DEVICE_TYPE RMT_PRXY (* Proxy for a Remotely Managed Device *)
  (* Standard: 61499 ITA; Description: Remotely Managed Device Proxy *)
  (* Version 0.2, 2002-01-01, JHC, Rockwell Automation, Added WAIT input. *)
  (* Version 0.1, 2001-01-21, JHC, Rockwell Automation, "Unencapsulated" DM_KRMT *)
  (* Version 0.0, 2000-12-31, JHC, Rockwell Automation, Initial version *)
  (* Compiler header: package fb.rt; import fb.rt.net.CLIENT_2_1; *)
  (* Compiler Java IBM VisualAge 3.0 *)
  VAR_INPUT
    MGR_ID : WSTRING := "localhost:61499"; (* Device manager socket ID *)
    WAIT : TIME := t#2s; (* Request timeout period *)
  END_VAR
  FBS
    MGR : DM_CLT;
    CLT : CLIENT_2_1;
  END_FBS
  EVENT_CONNECTIONS
    MGR.INITO TO CLT.INIT;
    CLT.INITO TO MGR.INIT;
    MGR.IND TO CLT.REQ;
    CLT.CNF TO MGR.RSP;
  END_CONNECTIONS
  DATA_CONNECTIONS
    MGR.QO TO CLT.QI;
    CLT.QO TO MGR.QI;
    MGR_ID TO CLT.ID;
    MGR.DST TO CLT.SD_1;
    MGR.RQST TO CLT.SD_2;
    CLT.RD_1 TO MGR.RESP;
    CLT.STATUS TO MGR.STATUS;
    WAIT TO MGR.WAIT;
  END_CONNECTIONS
END_DEVICE_TYPE
